// TIA Portal V19 export
FUNCTION_BLOCK "SpeedMachine_FB"   // FB36, LAD
TITLE = OPEN LOOP VELOCITY AXIS WTITH DRIVE S120 DRIVE TEL 1
// stored: Access Published, MemoryReserve 100, SetENOAutomatically false
   VAR_INPUT
      AreaInterface : "AreaInterface";
      ZSI : "udt_ZoneSafetyInterface";
      DSI : "udt_DeviceSafetyInterface";
      Drive : "TAx_DriveInterface";
      DataIn : "SpeedMachine_DataIn";
      CIn : "SpeedMachine_CIn";
      Config : "SpeedMachine_Config";
      HW_ID_TEL1 : HW_SUBMODULE;
   END_VAR
   VAR_OUTPUT
      MachineInterface : "MachineInterface";
      DataOut : "SpeedMachine_DataOut";
      COut : "SpeedMachine_COut";
   END_VAR
   VAR_IN_OUT
      Par : "SpeedMachine_Par";
      Warning : "SpeedMachine_Wng";
      Alarm : "SpeedMachine_Alr";
   END_VAR
   VAR
      Sts : Struct
         Standstill : Bool := TRUE;
         AlarmsPresence : Bool := FALSE;
         WarningsPresence : Bool := FALSE;
         Gen_Cnd : Bool;
         Bwd_Cnd : Bool := FALSE;
         Fwd_Cnd : Bool := FALSE;
         ReductionRatio : LReal := 1.0;   // mm / giro
      END_STRUCT;
      Ctrl : Struct
         StopDueDoorOpeningRequest : Bool;
         StopInPhase : Bool;
         StopProgrammed : Bool;
         StopAborting : Bool;
         Man_HighSpeed : Bool;
         Bwd_Man : Bool;
         Fwd_Man : Bool;
         Bwd_Aut : Bool;
         Fwd_Aut : Bool;
         Fan : Bool;
         Vel : LReal;
         Acc : LReal;
         Dec : LReal;
      END_STRUCT;
      Diag : Struct
         Drive : "TO_Diagnostic";
      END_STRUCT;
      S120 : "SpeedMotor";
      Fan_M : "Motor";
      TON_NoPendingCmd : IEC_TIMER;
      TON_Feed_DelayManChangeSpeed : IEC_TIMER;
      TON_MissingCndBwd { S7_SetPoint := 'True'} : IEC_TIMER;
      TON_MissingCndFwd { S7_SetPoint := 'True'} : IEC_TIMER;
      TON_Fan_DelayOff : IEC_TIMER;
      TON_Brake_TimeOut : IEC_TIMER;
      S120_STW_TEL1 { ExternalAccessible := 'False'; ExternalVisible := 'False'; ExternalWritable := 'False'} : PD_TEL1_IN;
      S120_ZSW_TEL1 { ExternalAccessible := 'False'; ExternalVisible := 'False'; ExternalWritable := 'False'} : PD_TEL1_OUT;
      GETIO_STW_TEL1 { S7_SetPoint := 'True'} : GETIO;
      SETIO_ZSW_TEL1 { S7_SetPoint := 'True'} : SETIO;
      AUX : Struct
         Bwd_Pb : Bool;
         Fwd_Pb : Bool;
      END_STRUCT;
      HMI : Struct
         Sts { S7_SetPoint := 'True'} : "UDT_HMI-Sts_SpeedMachineFB";
      END_STRUCT;
   END_VAR
   VAR_TEMP
      PE : Struct
         Bwd_Pb : Bool;
         Fwd_Pb : Bool;
      END_STRUCT;
      Req : Bool;
      VelMax_EngUnit : LReal;   // mm/min
      AccMax_EngUnit : LReal;   // mm/s²
      DecMax_EngUnit : LReal;   // mm/s²
      StandstillVelocity_RPM : LReal;
   END_VAR
   VAR_TEMP   // added for the SCL form of the ladder/FBD networks
      _w1 : Bool;
      _w2 : Bool;
   END_VAR
BEGIN

REGION Network 1 (SCL): Reset
   IF #AreaInterface.RstAlarms THEN

       #Alarm.BrakeTimeOut :=
       #Alarm.S120_ComErr :=

       #Warning.NotAutReady :=
       #Warning.MissingCnd_Bkw :=
       #Warning.MissingCnd_Fwd := FALSE;
   END_IF;
END_REGION

REGION Network 2: Alarm motor brake timeout
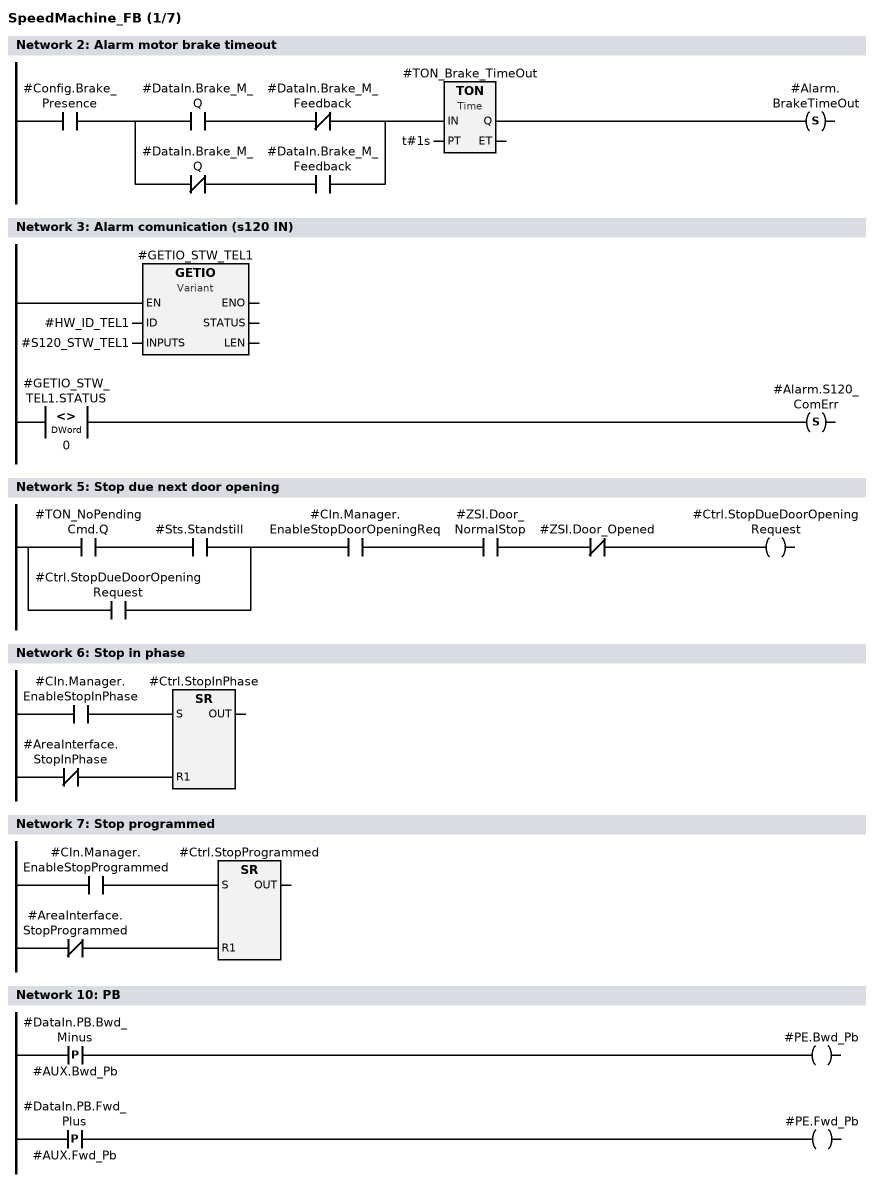
   RUNG wire#powerrail
      Contact( #Config.Brake_Presence )
      wire#w1
      Contact( #DataIn.Brake_M_Q )
      I_Contact( #DataIn.Brake_M_Feedback )
      wire#w2
      { S7_Templates := "time_type := Time" } #TON_Brake_TimeOut.TON(pt := t#1s, et =>)
      S_Coil( #Alarm.BrakeTimeOut )
   END_RUNG
   RUNG wire#w1
      I_Contact( #DataIn.Brake_M_Q )
      Contact( #DataIn.Brake_M_Feedback )
   END_RUNG wire#w2
   // the same network as SCL:
   #TON_Brake_TimeOut.TON(IN := #Config.Brake_Presence AND ((#DataIn.Brake_M_Q AND NOT #DataIn.Brake_M_Feedback) OR (NOT #DataIn.Brake_M_Q AND #DataIn.Brake_M_Feedback)),
                          PT := t#1s);
   IF #TON_Brake_TimeOut.Q THEN #Alarm.BrakeTimeOut := TRUE; END_IF;
END_REGION

REGION Network 3: Alarm comunication (s120 IN)
   RUNG wire#powerrail
      { S7_Templates := "[ptr_type := Variant, id_type := HW_SUBMODULE]" } #GETIO_STW_TEL1.GETIO(ID := #HW_ID_TEL1, INPUTS := #S120_STW_TEL1, STATUS =>, LEN =>)
   END_RUNG
   RUNG wire#powerrail
      { S7_Templates := "SrcType := DWord" } NE_Contact(in1 := #GETIO_STW_TEL1.STATUS, in2 := 0)
      S_Coil( #Alarm.S120_ComErr )
   END_RUNG
   // the same network as SCL:
   #GETIO_STW_TEL1(ID := #HW_ID_TEL1, INPUTS := #S120_STW_TEL1);   // GETIO
   IF #GETIO_STW_TEL1.STATUS <> 0 THEN #Alarm.S120_ComErr := TRUE; END_IF;
END_REGION

REGION Network 4: <<< MACHINE STOP >>>
END_REGION

REGION Network 5: Stop due next door opening
   RUNG wire#powerrail
      Contact( #TON_NoPendingCmd.Q )
      Contact( #Sts.Standstill )
      wire#w1
      Contact( #CIn.Manager.EnableStopDoorOpeningReq )
      Contact( #ZSI.Door_NormalStop )
      I_Contact( #ZSI.Door_Opened )
      Coil( #Ctrl.StopDueDoorOpeningRequest )
   END_RUNG
   RUNG wire#powerrail
      Contact( #Ctrl.StopDueDoorOpeningRequest )
   END_RUNG wire#w1
   // the same network as SCL:
   #Ctrl.StopDueDoorOpeningRequest := ((#TON_NoPendingCmd.Q AND #Sts.Standstill) OR #Ctrl.StopDueDoorOpeningRequest) AND #CIn.Manager.EnableStopDoorOpeningReq AND #ZSI.Door_NormalStop AND NOT #ZSI.Door_Opened;
END_REGION

REGION Network 6: Stop in phase
   RUNG wire#powerrail
      Contact( #CIn.Manager.EnableStopInPhase )
      S_SR(operand := #Ctrl.StopInPhase, r1 := wire#w1)
   END_RUNG
   RUNG wire#powerrail
      I_Contact( #AreaInterface.StopInPhase )
   END_RUNG wire#w1
   // the same network as SCL:
   IF #CIn.Manager.EnableStopInPhase THEN
       #Ctrl.StopInPhase := TRUE;   // SR flip-flop
   END_IF;
   IF NOT #AreaInterface.StopInPhase THEN #Ctrl.StopInPhase := FALSE; END_IF;
END_REGION

REGION Network 7: Stop programmed
   RUNG wire#powerrail
      Contact( #CIn.Manager.EnableStopProgrammed )
      S_SR(operand := #Ctrl.StopProgrammed, r1 := wire#w1)
   END_RUNG
   RUNG wire#powerrail
      I_Contact( #AreaInterface.StopProgrammed )
   END_RUNG wire#w1
   // the same network as SCL:
   IF #CIn.Manager.EnableStopProgrammed THEN
       #Ctrl.StopProgrammed := TRUE;   // SR flip-flop
   END_IF;
   IF NOT #AreaInterface.StopProgrammed THEN #Ctrl.StopProgrammed := FALSE; END_IF;
END_REGION

REGION Network 8: >
END_REGION

REGION Network 9: <<< FEED >>>
END_REGION

REGION Network 10: PB
   RUNG wire#powerrail
      P_Contact(operand := #DataIn.PB.Bwd_Minus, bit := #AUX.Bwd_Pb)
      Coil( #PE.Bwd_Pb )
   END_RUNG
   RUNG wire#powerrail
      P_Contact(operand := #DataIn.PB.Fwd_Plus, bit := #AUX.Fwd_Pb)
      Coil( #PE.Fwd_Pb )
   END_RUNG
   // the same network as SCL:
   #_w1 := #DataIn.PB.Bwd_Minus AND NOT #AUX.Bwd_Pb;   // rising edge of #DataIn.PB.Bwd_Minus
   #AUX.Bwd_Pb := #DataIn.PB.Bwd_Minus;
   #PE.Bwd_Pb := #_w1;
   #_w2 := #DataIn.PB.Fwd_Plus AND NOT #AUX.Fwd_Pb;   // rising edge of #DataIn.PB.Fwd_Plus
   #AUX.Fwd_Pb := #DataIn.PB.Fwd_Plus;
   #PE.Fwd_Pb := #_w2;
END_REGION

REGION Network 11: Man
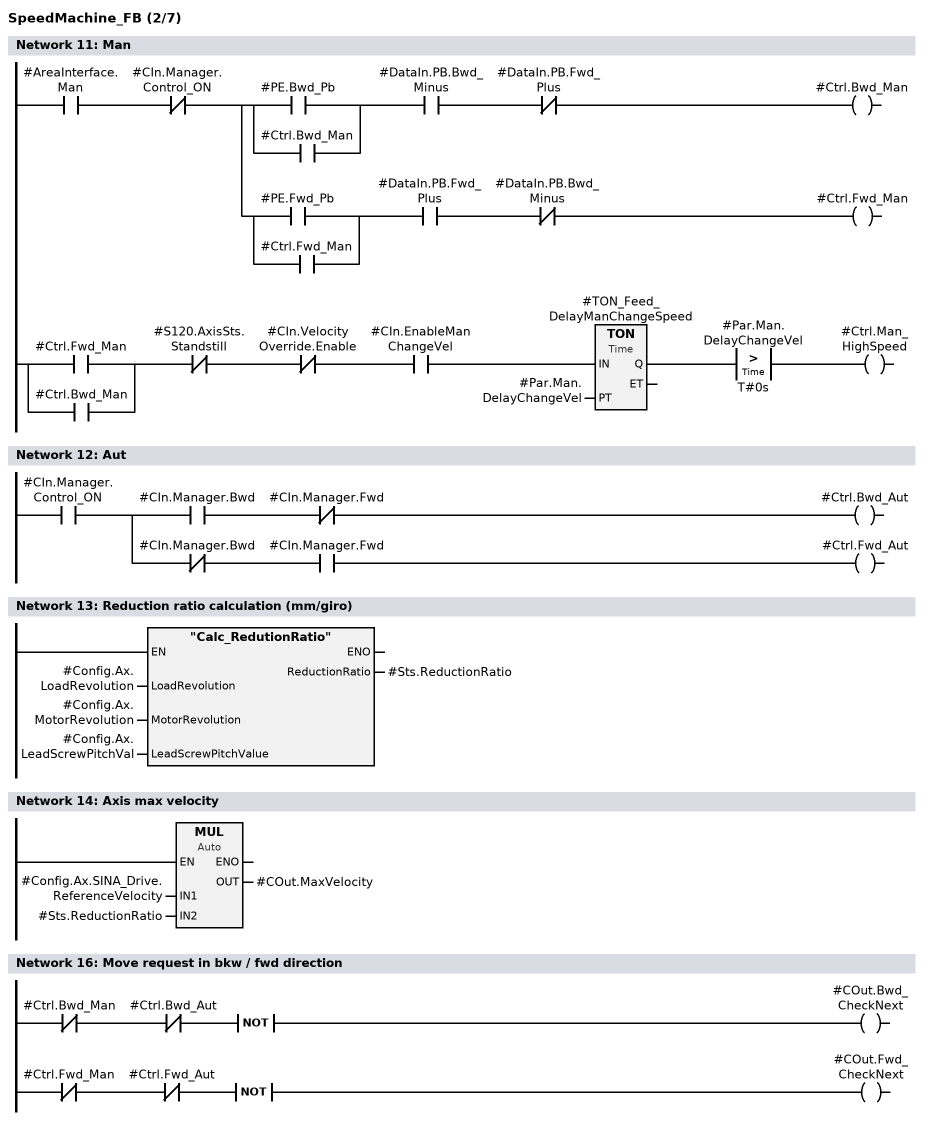
   RUNG wire#powerrail
      Contact( #AreaInterface.Man )
      I_Contact( #CIn.Manager.Control_ON )
      wire#w1
      Contact( #PE.Bwd_Pb )
      wire#w2
      Contact( #DataIn.PB.Bwd_Minus )
      I_Contact( #DataIn.PB.Fwd_Plus )
      Coil( #Ctrl.Bwd_Man )
   END_RUNG
   RUNG wire#w1
      Contact( #Ctrl.Bwd_Man )
   END_RUNG wire#w2
   RUNG wire#w1
      Contact( #PE.Fwd_Pb )
      wire#w3
      Contact( #DataIn.PB.Fwd_Plus )
      I_Contact( #DataIn.PB.Bwd_Minus )
      Coil( #Ctrl.Fwd_Man )
   END_RUNG
   RUNG wire#w1
      Contact( #Ctrl.Fwd_Man )
   END_RUNG wire#w3
   RUNG wire#powerrail
      Contact( #Ctrl.Fwd_Man )
      wire#w4
      I_Contact( #S120.AxisSts.Standstill )
      I_Contact( #CIn.VelocityOverride.Enable )
      Contact( #CIn.EnableManChangeVel )
      { S7_Templates := "time_type := Time" } #TON_Feed_DelayManChangeSpeed.TON(pt := #Par.Man.DelayChangeVel, et =>)
      { S7_Templates := "SrcType := Time" } GT_Contact(in1 := #Par.Man.DelayChangeVel, in2 := T#0s)
      Coil( #Ctrl.Man_HighSpeed )
   END_RUNG
   RUNG wire#powerrail
      Contact( #Ctrl.Bwd_Man )
   END_RUNG wire#w4
   // the same network as SCL:
   #_w1 := #AreaInterface.Man AND NOT #CIn.Manager.Control_ON;
   #Ctrl.Bwd_Man := #_w1 AND (#PE.Bwd_Pb OR #Ctrl.Bwd_Man) AND #DataIn.PB.Bwd_Minus AND NOT #DataIn.PB.Fwd_Plus;
   #Ctrl.Fwd_Man := #_w1 AND (#PE.Fwd_Pb OR #Ctrl.Fwd_Man) AND #DataIn.PB.Fwd_Plus AND NOT #DataIn.PB.Bwd_Minus;
   #TON_Feed_DelayManChangeSpeed.TON(IN := (#Ctrl.Fwd_Man OR #Ctrl.Bwd_Man) AND NOT #S120.AxisSts.Standstill AND NOT #CIn.VelocityOverride.Enable AND #CIn.EnableManChangeVel,
                           PT := #Par.Man.DelayChangeVel);
   #Ctrl.Man_HighSpeed := #TON_Feed_DelayManChangeSpeed.Q AND (#Par.Man.DelayChangeVel > T#0s);
END_REGION

REGION Network 12: Aut
   RUNG wire#powerrail
      Contact( #CIn.Manager.Control_ON )
      wire#w1
      Contact( #CIn.Manager.Bwd )
      I_Contact( #CIn.Manager.Fwd )
      Coil( #Ctrl.Bwd_Aut )
   END_RUNG
   RUNG wire#w1
      I_Contact( #CIn.Manager.Bwd )
      Contact( #CIn.Manager.Fwd )
      Coil( #Ctrl.Fwd_Aut )
   END_RUNG
   // the same network as SCL:
   #Ctrl.Bwd_Aut := #CIn.Manager.Control_ON AND #CIn.Manager.Bwd AND NOT #CIn.Manager.Fwd;
   #Ctrl.Fwd_Aut := #CIn.Manager.Control_ON AND NOT #CIn.Manager.Bwd AND #CIn.Manager.Fwd;
END_REGION

REGION Network 13: Reduction ratio calculation (mm/giro)
   RUNG wire#powerrail
      "Calc_RedutionRatio"(LoadRevolution := #Config.Ax.LoadRevolution, MotorRevolution := #Config.Ax.MotorRevolution, LeadScrewPitchValue := #Config.Ax.LeadScrewPitchVal, ReductionRatio => #Sts.ReductionRatio)
   END_RUNG
   // the same network as SCL:
   "Calc_RedutionRatio"(LoadRevolution := #Config.Ax.LoadRevolution,
                        MotorRevolution := #Config.Ax.MotorRevolution,
                        LeadScrewPitchValue := #Config.Ax.LeadScrewPitchVal,
                        ReductionRatio => #Sts.ReductionRatio);
END_REGION

REGION Network 14: Axis max velocity
   RUNG wire#powerrail
      Mul(in1 := #Config.Ax.SINA_Drive.ReferenceVelocity, in2 := #Sts.ReductionRatio, out => #COut.MaxVelocity)
   END_RUNG
   // the same network as SCL:
   #COut.MaxVelocity := #Config.Ax.SINA_Drive.ReferenceVelocity * #Sts.ReductionRatio;
END_REGION

REGION Network 15 (SCL): Velocity & Dynamics
   #VelMax_EngUnit := #Config.Ax.SINA_Drive.ReferenceVelocity *  #Sts.ReductionRatio;
   #AccMax_EngUnit := (#Config.Ax.SINA_Drive.ReferenceVelocity / 60.0 / #Config.Ax.MinAccTime) * #Sts.ReductionRatio; // Giri/s² * mm/Giro = mm/s²
   #DecMax_EngUnit := (#Config.Ax.SINA_Drive.ReferenceVelocity / 60.0 / #Config.Ax.MinDecTime) * #Sts.ReductionRatio; // Giri/s² * mm/Giro = mm/s²


   #Ctrl.Vel := 0.0;

   IF #Ctrl.Bwd_Man AND #S120.AxisCtrl.MoveMinus THEN


       #Ctrl.Acc := #Par.Man.Acc;
       #Ctrl.Dec := #Par.Man.Dec;

       IF #Ctrl.Man_HighSpeed THEN
           #Ctrl.Vel := #Par.Man.VelBwd;
       ELSE
           #Ctrl.Vel := #Par.Man.VelFwdLow;
       END_IF;

   ELSIF #Ctrl.Fwd_Man AND #S120.AxisCtrl.MovePlus THEN


       #Ctrl.Acc := #Par.Man.Acc;
       #Ctrl.Dec := #Par.Man.Dec;

       IF #Ctrl.Man_HighSpeed THEN
           #Ctrl.Vel := #Par.Man.VelFwdHigh;
       ELSE
           #Ctrl.Vel := #Par.Man.VelFwdLow;
       END_IF;


   ELSIF (#Ctrl.Bwd_Aut AND #S120.AxisCtrl.MoveMinus) OR (#Ctrl.Fwd_Aut AND #S120.AxisCtrl.MovePlus)  THEN

       #Ctrl.Vel := #CIn.Manager.Vel;
       #Ctrl.Acc := #CIn.Manager.Acc;
       #Ctrl.Dec := #CIn.Manager.Dec;

   END_IF;



   // Dynamics limit
   #Ctrl.Vel := MIN(IN1:= #Ctrl.Vel,IN2:= #VelMax_EngUnit);


   #Ctrl.Acc := MIN(IN1:= #Ctrl.Acc,IN2:= #AccMax_EngUnit);

   IF #Ctrl.Acc <= 0.0 THEN
       #Ctrl.Acc := #Par.Man.Acc;
   END_IF;

   #Ctrl.Dec := MIN(IN1:= #Ctrl.Dec,IN2:= #DecMax_EngUnit);
   IF #Ctrl.Dec <= 0.0 THEN
       #Ctrl.Dec := #Par.Man.Dec;
   END_IF;





   // SLS velocity limit
   //
   IF #ZSI.Door_Opened AND #Ctrl.Vel > #Config.SLS_VEL THEN
       #Ctrl.Vel := #Config.SLS_VEL;
   END_IF;


   // Brake not open... Velocity  = 0.0
   // 
   IF #Config.Brake_Presence AND NOT #DataIn.Brake_M_Feedback THEN
       #S120.AxisCtrl.Velocity := 0.0;
   END_IF;



   // Conversion and write dynamics value
   // 
   #S120.AxisCtrl.Velocity := #Ctrl.Vel / #Sts.ReductionRatio; // mm/minuto -> giri/minuto

   // Velocity override
   // 
   IF #CIn.VelocityOverride.Enable THEN

       #S120.AxisCtrl.Velocity := #S120.AxisCtrl.Velocity  * (LIMIT(MN := 1.0, IN := #CIn.VelocityOverride.Value, MX := 200.0)/100);
   END_IF;



   #S120.AxisCtrl.Acceleration := #Ctrl.Acc / #Sts.ReductionRatio; // mm/s2 -> giri/s²
   #S120.AxisCtrl.Deceleration := #Ctrl.Dec / #Sts.ReductionRatio; // mm/s2 -> giri/s²


   //#StandstillVelocity_RPM := #Config.Ax.StandstillVelocity / #Sts.ReductionRatio;
END_REGION

REGION Network 16: Move request in bkw / fwd direction
   RUNG wire#powerrail
      I_Contact( #Ctrl.Bwd_Man )
      I_Contact( #Ctrl.Bwd_Aut )
      Not()
      Coil( #COut.Bwd_CheckNext )
   END_RUNG
   RUNG wire#powerrail
      I_Contact( #Ctrl.Fwd_Man )
      I_Contact( #Ctrl.Fwd_Aut )
      Not()
      Coil( #COut.Fwd_CheckNext )
   END_RUNG
   // the same network as SCL:
   #COut.Bwd_CheckNext := NOT (NOT #Ctrl.Bwd_Man AND NOT #Ctrl.Bwd_Aut);
   #COut.Fwd_CheckNext := NOT (NOT #Ctrl.Fwd_Man AND NOT #Ctrl.Fwd_Aut);
END_REGION

REGION Network 17: Conditions
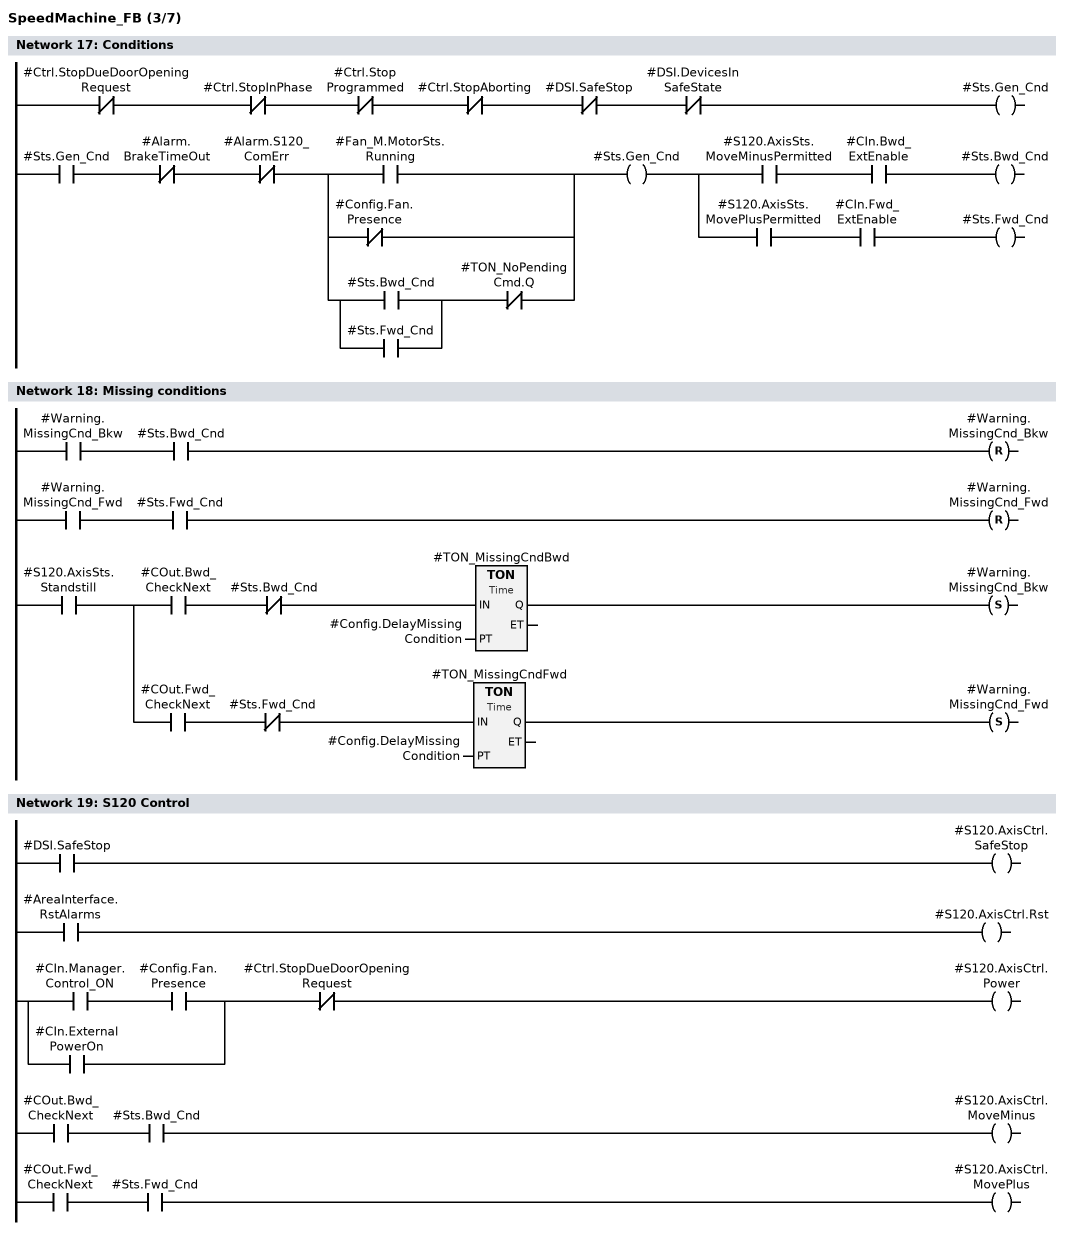
   RUNG wire#powerrail
      I_Contact( #Ctrl.StopDueDoorOpeningRequest )
      I_Contact( #Ctrl.StopInPhase )
      I_Contact( #Ctrl.StopProgrammed )
      I_Contact( #Ctrl.StopAborting )
      I_Contact( #DSI.SafeStop )
      I_Contact( #DSI.DevicesInSafeState )
      Coil( #Sts.Gen_Cnd )
   END_RUNG
   RUNG wire#powerrail
      Contact( #Sts.Gen_Cnd )
      I_Contact( #Alarm.BrakeTimeOut )
      I_Contact( #Alarm.S120_ComErr )
      wire#w1
      Contact( #Fan_M.MotorSts.Running )
      wire#w2
      Coil( #Sts.Gen_Cnd )
      wire#w4
      Contact( #S120.AxisSts.MoveMinusPermitted )
      Contact( #CIn.Bwd_ExtEnable )
      Coil( #Sts.Bwd_Cnd )
   END_RUNG
   RUNG wire#w1
      I_Contact( #Config.Fan.Presence )
   END_RUNG wire#w2
   RUNG wire#w1
      Contact( #Sts.Bwd_Cnd )
      wire#w3
      I_Contact( #TON_NoPendingCmd.Q )
   END_RUNG wire#w2
   RUNG wire#w1
      Contact( #Sts.Fwd_Cnd )
   END_RUNG wire#w3
   RUNG wire#w4
      Contact( #S120.AxisSts.MovePlusPermitted )
      Contact( #CIn.Fwd_ExtEnable )
      Coil( #Sts.Fwd_Cnd )
   END_RUNG
   // the same network as SCL:
   #Sts.Gen_Cnd := NOT #Ctrl.StopDueDoorOpeningRequest AND NOT #Ctrl.StopInPhase AND NOT #Ctrl.StopProgrammed AND NOT #Ctrl.StopAborting AND NOT #DSI.SafeStop AND NOT #DSI.DevicesInSafeState;
   #Sts.Gen_Cnd := #Sts.Gen_Cnd AND NOT #Alarm.BrakeTimeOut AND NOT #Alarm.S120_ComErr AND (#Fan_M.MotorSts.Running OR NOT #Config.Fan.Presence OR ((#Sts.Bwd_Cnd OR #Sts.Fwd_Cnd) AND NOT #TON_NoPendingCmd.Q));
   #Sts.Bwd_Cnd := #Sts.Gen_Cnd AND #S120.AxisSts.MoveMinusPermitted AND #CIn.Bwd_ExtEnable;
   #Sts.Fwd_Cnd := #Sts.Gen_Cnd AND #S120.AxisSts.MovePlusPermitted AND #CIn.Fwd_ExtEnable;
END_REGION

REGION Network 18: Missing conditions
   RUNG wire#powerrail
      Contact( #Warning.MissingCnd_Bkw )
      Contact( #Sts.Bwd_Cnd )
      R_Coil( #Warning.MissingCnd_Bkw )
   END_RUNG
   RUNG wire#powerrail
      Contact( #Warning.MissingCnd_Fwd )
      Contact( #Sts.Fwd_Cnd )
      R_Coil( #Warning.MissingCnd_Fwd )
   END_RUNG
   RUNG wire#powerrail
      Contact( #S120.AxisSts.Standstill )
      wire#w1
      Contact( #COut.Bwd_CheckNext )
      I_Contact( #Sts.Bwd_Cnd )
      { S7_Templates := "time_type := Time" } #TON_MissingCndBwd.TON(pt := #Config.DelayMissingCondition, et =>)
      S_Coil( #Warning.MissingCnd_Bkw )
   END_RUNG
   RUNG wire#w1
      Contact( #COut.Fwd_CheckNext )
      I_Contact( #Sts.Fwd_Cnd )
      { S7_Templates := "time_type := Time" } #TON_MissingCndFwd.TON(pt := #Config.DelayMissingCondition, et =>)
      S_Coil( #Warning.MissingCnd_Fwd )
   END_RUNG
   // the same network as SCL:
   IF #Warning.MissingCnd_Bkw AND #Sts.Bwd_Cnd THEN #Warning.MissingCnd_Bkw := FALSE; END_IF;
   IF #Warning.MissingCnd_Fwd AND #Sts.Fwd_Cnd THEN #Warning.MissingCnd_Fwd := FALSE; END_IF;
   #TON_MissingCndBwd.TON(IN := #S120.AxisSts.Standstill AND #COut.Bwd_CheckNext AND NOT #Sts.Bwd_Cnd,
                          PT := #Config.DelayMissingCondition);
   IF #TON_MissingCndBwd.Q THEN #Warning.MissingCnd_Bkw := TRUE; END_IF;
   #TON_MissingCndFwd.TON(IN := #S120.AxisSts.Standstill AND #COut.Fwd_CheckNext AND NOT #Sts.Fwd_Cnd,
                          PT := #Config.DelayMissingCondition);
   IF #TON_MissingCndFwd.Q THEN #Warning.MissingCnd_Fwd := TRUE; END_IF;
END_REGION

REGION Network 19: S120 Control
   RUNG wire#powerrail
      Contact( #DSI.SafeStop )
      Coil( #S120.AxisCtrl.SafeStop )
   END_RUNG
   RUNG wire#powerrail
      Contact( #AreaInterface.RstAlarms )
      Coil( #S120.AxisCtrl.Rst )
   END_RUNG
   RUNG wire#powerrail
      Contact( #CIn.Manager.Control_ON )
      Contact( #Config.Fan.Presence )
      wire#w1
      I_Contact( #Ctrl.StopDueDoorOpeningRequest )
      Coil( #S120.AxisCtrl.Power )
   END_RUNG
   RUNG wire#powerrail
      Contact( #CIn.ExternalPowerOn )
   END_RUNG wire#w1
   RUNG wire#powerrail
      Contact( #COut.Bwd_CheckNext )
      Contact( #Sts.Bwd_Cnd )
      Coil( #S120.AxisCtrl.MoveMinus )
   END_RUNG
   RUNG wire#powerrail
      Contact( #COut.Fwd_CheckNext )
      Contact( #Sts.Fwd_Cnd )
      Coil( #S120.AxisCtrl.MovePlus )
   END_RUNG
   // the same network as SCL:
   #S120.AxisCtrl.SafeStop := #DSI.SafeStop;
   #S120.AxisCtrl.Rst := #AreaInterface.RstAlarms;
   #S120.AxisCtrl.Power := ((#CIn.Manager.Control_ON AND #Config.Fan.Presence) OR #CIn.ExternalPowerOn) AND NOT #Ctrl.StopDueDoorOpeningRequest;
   #S120.AxisCtrl.MoveMinus := #COut.Bwd_CheckNext AND #Sts.Bwd_Cnd;
   #S120.AxisCtrl.MovePlus := #COut.Fwd_CheckNext AND #Sts.Fwd_Cnd;
END_REGION

REGION Network 20: S120 manager
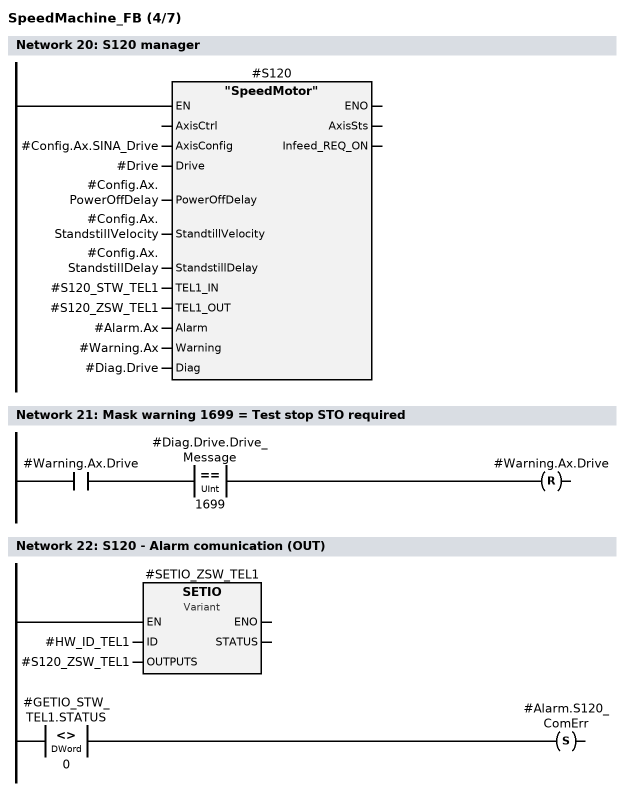
   RUNG wire#powerrail
      #S120(AxisCtrl :=, AxisConfig := #Config.Ax.SINA_Drive, Drive := #Drive, PowerOffDelay := #Config.Ax.PowerOffDelay, StandtillVelocity := #Config.Ax.StandstillVelocity, StandstillDelay := #Config.Ax.StandstillDelay, TEL1_IN := #S120_STW_TEL1, TEL1_OUT := #S120_ZSW_TEL1, Alarm := #Alarm.Ax, Warning := #Warning.Ax, Diag := #Diag.Drive, AxisSts =>, Infeed_REQ_ON =>)
   END_RUNG
   // the same network as SCL:
   #S120(AxisConfig := #Config.Ax.SINA_Drive,   // "SpeedMotor"
         Drive := #Drive,
         PowerOffDelay := #Config.Ax.PowerOffDelay,
         StandtillVelocity := #Config.Ax.StandstillVelocity,
         StandstillDelay := #Config.Ax.StandstillDelay,
         TEL1_IN := #S120_STW_TEL1,
         TEL1_OUT := #S120_ZSW_TEL1,
         Alarm := #Alarm.Ax,
         Warning := #Warning.Ax,
         Diag := #Diag.Drive);
END_REGION

REGION Network 21: Mask warning 1699 = Test stop STO required
   RUNG wire#powerrail
      Contact( #Warning.Ax.Drive )
      { S7_Templates := "SrcType := UInt" } EQ_Contact(in1 := #Diag.Drive.Drive_Message, in2 := 1699)
      R_Coil( #Warning.Ax.Drive )
   END_RUNG
   // the same network as SCL:
   IF #Warning.Ax.Drive AND (#Diag.Drive.Drive_Message = 1699) THEN #Warning.Ax.Drive := FALSE; END_IF;
END_REGION

REGION Network 22: S120 - Alarm comunication (OUT)
   RUNG wire#powerrail
      { S7_Templates := "[card := 0, ptr_type := Variant, id_type := HW_SUBMODULE]" } #SETIO_ZSW_TEL1.SETIO(ID := #HW_ID_TEL1, OUTPUTS := #S120_ZSW_TEL1, STATUS =>)
   END_RUNG
   RUNG wire#powerrail
      { S7_Templates := "SrcType := DWord" } NE_Contact(in1 := #GETIO_STW_TEL1.STATUS, in2 := 0)
      S_Coil( #Alarm.S120_ComErr )
   END_RUNG
   // the same network as SCL:
   #SETIO_ZSW_TEL1(ID := #HW_ID_TEL1, OUTPUTS := #S120_ZSW_TEL1);   // SETIO
   IF #GETIO_STW_TEL1.STATUS <> 0 THEN #Alarm.S120_ComErr := TRUE; END_IF;
END_REGION

REGION Network 23: Coordination Out
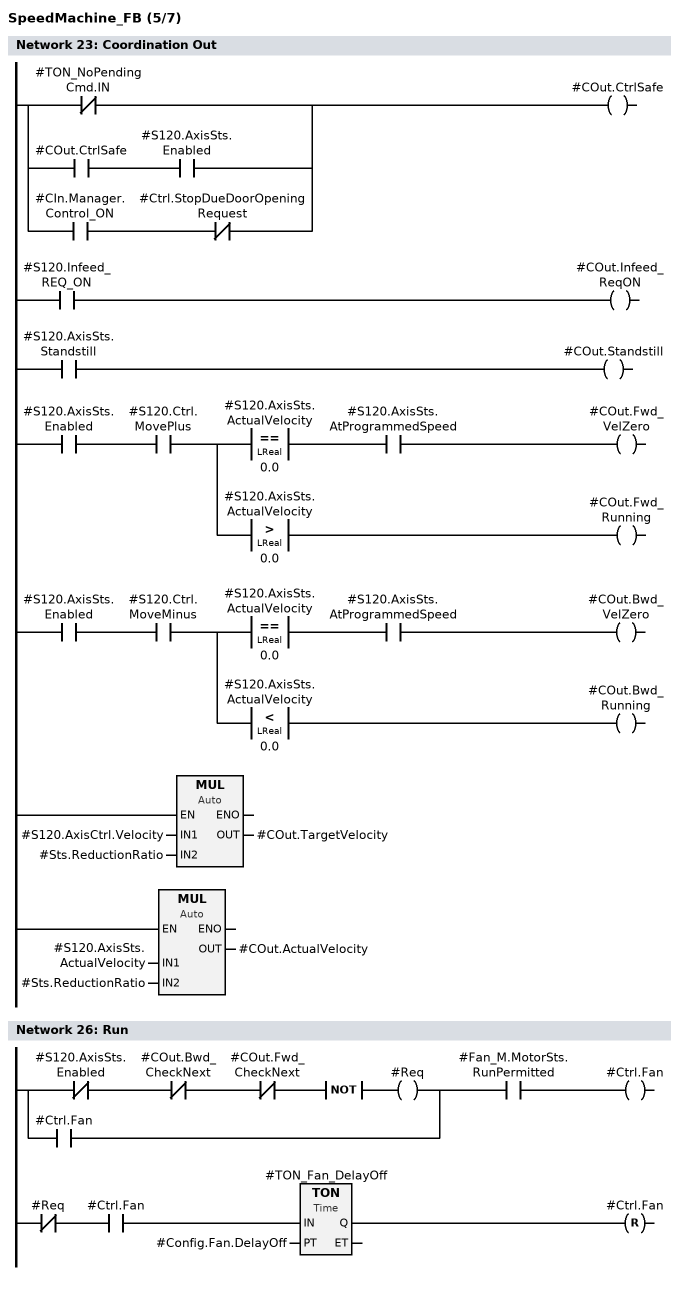
   RUNG wire#powerrail
      I_Contact( #TON_NoPendingCmd.IN )
      wire#w1
      Coil( #COut.CtrlSafe )
   END_RUNG
   RUNG wire#powerrail
      Contact( #COut.CtrlSafe )
      Contact( #S120.AxisSts.Enabled )
   END_RUNG wire#w1
   RUNG wire#powerrail
      Contact( #CIn.Manager.Control_ON )
      I_Contact( #Ctrl.StopDueDoorOpeningRequest )
   END_RUNG wire#w1
   RUNG wire#powerrail
      Contact( #S120.Infeed_REQ_ON )
      Coil( #COut.Infeed_ReqON )
   END_RUNG
   RUNG wire#powerrail
      Contact( #S120.AxisSts.Standstill )
      Coil( #COut.Standstill )
   END_RUNG
   RUNG wire#powerrail
      Contact( #S120.AxisSts.Enabled )
      Contact( #S120.Ctrl.MovePlus )
      wire#w2
      { S7_Templates := "SrcType := LReal" } EQ_Contact(in1 := #S120.AxisSts.ActualVelocity, in2 := 0.0)
      Contact( #S120.AxisSts.AtProgrammedSpeed )
      Coil( #COut.Fwd_VelZero )
   END_RUNG
   RUNG wire#w2
      { S7_Templates := "SrcType := LReal" } GT_Contact(in1 := #S120.AxisSts.ActualVelocity, in2 := 0.0)
      Coil( #COut.Fwd_Running )
   END_RUNG
   RUNG wire#powerrail
      Contact( #S120.AxisSts.Enabled )
      Contact( #S120.Ctrl.MoveMinus )
      wire#w3
      { S7_Templates := "SrcType := LReal" } EQ_Contact(in1 := #S120.AxisSts.ActualVelocity, in2 := 0.0)
      Contact( #S120.AxisSts.AtProgrammedSpeed )
      Coil( #COut.Bwd_VelZero )
   END_RUNG
   RUNG wire#w3
      { S7_Templates := "SrcType := LReal" } LT_Contact(in1 := #S120.AxisSts.ActualVelocity, in2 := 0.0)
      Coil( #COut.Bwd_Running )
   END_RUNG
   RUNG wire#powerrail
      { S7_GenerateENO := "TRUE" } Mul(in1 := #S120.AxisCtrl.Velocity, in2 := #Sts.ReductionRatio, out => #COut.TargetVelocity)
   END_RUNG
   RUNG wire#powerrail
      { S7_GenerateENO := "TRUE" } Mul(in1 := #S120.AxisSts.ActualVelocity, in2 := #Sts.ReductionRatio, out => #COut.ActualVelocity)
   END_RUNG
   // the same network as SCL:
   #COut.CtrlSafe := NOT #TON_NoPendingCmd.IN OR (#COut.CtrlSafe AND #S120.AxisSts.Enabled) OR (#CIn.Manager.Control_ON AND NOT #Ctrl.StopDueDoorOpeningRequest);
   #COut.Infeed_ReqON := #S120.Infeed_REQ_ON;
   #COut.Standstill := #S120.AxisSts.Standstill;
   #_w1 := #S120.AxisSts.Enabled AND #S120.Ctrl.MovePlus;
   #COut.Fwd_VelZero := #_w1 AND (#S120.AxisSts.ActualVelocity = 0.0) AND #S120.AxisSts.AtProgrammedSpeed;
   #COut.Fwd_Running := #_w1 AND (#S120.AxisSts.ActualVelocity > 0.0);
   #_w2 := #S120.AxisSts.Enabled AND #S120.Ctrl.MoveMinus;
   #COut.Bwd_VelZero := #_w2 AND (#S120.AxisSts.ActualVelocity = 0.0) AND #S120.AxisSts.AtProgrammedSpeed;
   #COut.Bwd_Running := #_w2 AND (#S120.AxisSts.ActualVelocity < 0.0);
   #COut.TargetVelocity := #S120.AxisCtrl.Velocity * #Sts.ReductionRatio;
   #COut.ActualVelocity := #S120.AxisSts.ActualVelocity * #Sts.ReductionRatio;
END_REGION

REGION Network 24: >
END_REGION

REGION Network 25: <<< MOTOR FAN >>>
END_REGION

REGION Network 26: Run
   RUNG wire#powerrail
      I_Contact( #S120.AxisSts.Enabled )
      I_Contact( #COut.Bwd_CheckNext )
      I_Contact( #COut.Fwd_CheckNext )
      Not()
      Coil( #Req )
      wire#w1
      Contact( #Fan_M.MotorSts.RunPermitted )
      Coil( #Ctrl.Fan )
   END_RUNG
   RUNG wire#powerrail
      Contact( #Ctrl.Fan )
   END_RUNG wire#w1
   RUNG wire#powerrail
      I_Contact( #Req )
      Contact( #Ctrl.Fan )
      { S7_Templates := "time_type := Time" } #TON_Fan_DelayOff.TON(pt := #Config.Fan.DelayOff, et =>)
      R_Coil( #Ctrl.Fan )
   END_RUNG
   // the same network as SCL:
   #Req := NOT (NOT #S120.AxisSts.Enabled AND NOT #COut.Bwd_CheckNext AND NOT #COut.Fwd_CheckNext);
   #Ctrl.Fan := (#Req OR #Ctrl.Fan) AND #Fan_M.MotorSts.RunPermitted;
   #TON_Fan_DelayOff.TON(IN := NOT #Req AND #Ctrl.Fan, PT := #Config.Fan.DelayOff);
   IF #TON_Fan_DelayOff.Q THEN #Ctrl.Fan := FALSE; END_IF;
END_REGION

REGION Network 27: Device
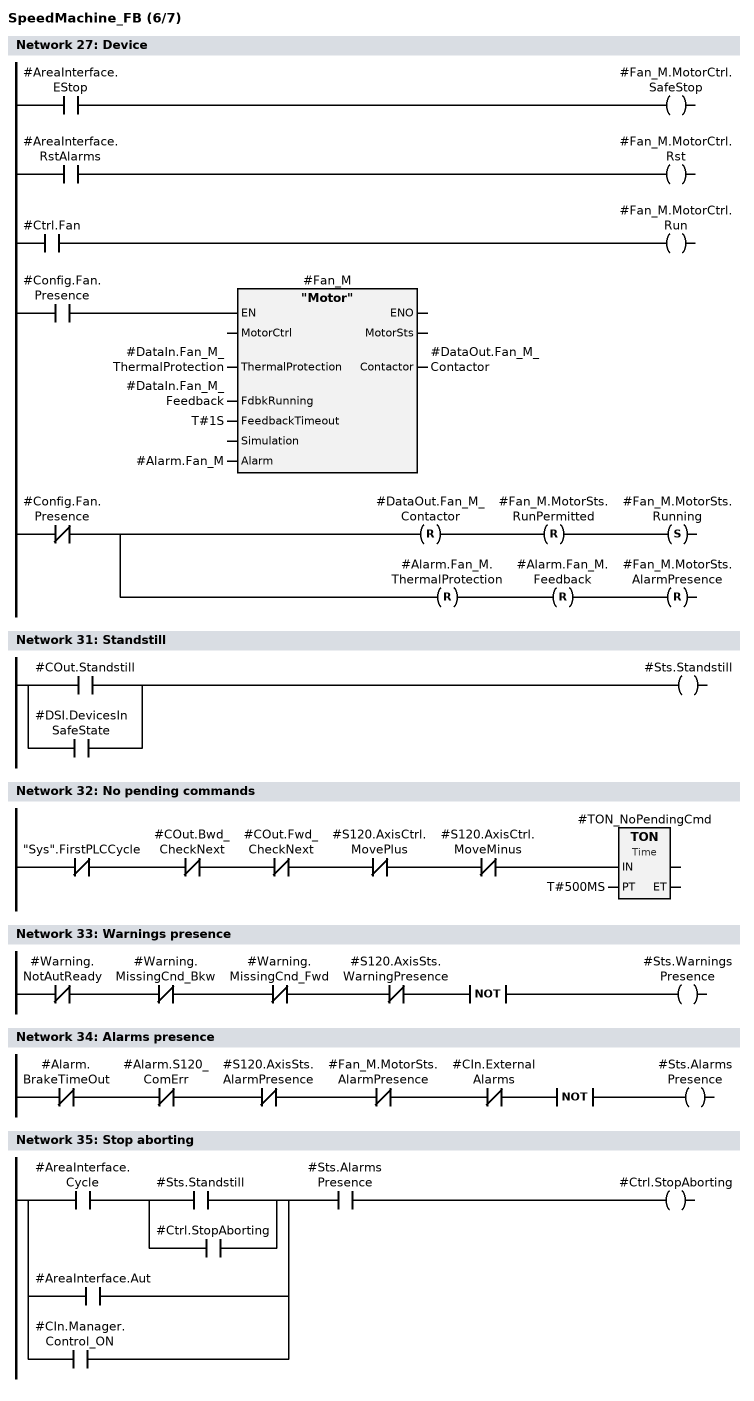
   RUNG wire#powerrail
      Contact( #AreaInterface.EStop )
      Coil( #Fan_M.MotorCtrl.SafeStop )
   END_RUNG
   RUNG wire#powerrail
      Contact( #AreaInterface.RstAlarms )
      Coil( #Fan_M.MotorCtrl.Rst )
   END_RUNG
   RUNG wire#powerrail
      Contact( #Ctrl.Fan )
      Coil( #Fan_M.MotorCtrl.Run )
   END_RUNG
   RUNG wire#powerrail
      Contact( #Config.Fan.Presence )
      #Fan_M(MotorCtrl :=, ThermalProtection := #DataIn.Fan_M_ThermalProtection, FdbkRunning := #DataIn.Fan_M_Feedback, FeedbackTimeout := T#1S, Simulation :=, Alarm := #Alarm.Fan_M, MotorSts =>, Contactor => #DataOut.Fan_M_Contactor)
   END_RUNG
   RUNG wire#powerrail
      I_Contact( #Config.Fan.Presence )
      wire#w1
      R_Coil( #DataOut.Fan_M_Contactor )
      R_Coil( #Fan_M.MotorSts.RunPermitted )
      S_Coil( #Fan_M.MotorSts.Running )
   END_RUNG
   RUNG wire#w1
      R_Coil( #Alarm.Fan_M.ThermalProtection )
      R_Coil( #Alarm.Fan_M.Feedback )
      R_Coil( #Fan_M.MotorSts.AlarmPresence )
   END_RUNG
   // the same network as SCL:
   #Fan_M.MotorCtrl.SafeStop := #AreaInterface.EStop;
   #Fan_M.MotorCtrl.Rst := #AreaInterface.RstAlarms;
   #Fan_M.MotorCtrl.Run := #Ctrl.Fan;
   IF #Config.Fan.Presence THEN
       #Fan_M(ThermalProtection := #DataIn.Fan_M_ThermalProtection,   // "Motor"
              FdbkRunning := #DataIn.Fan_M_Feedback,
              FeedbackTimeout := T#1S,
              Alarm := #Alarm.Fan_M,
              Contactor => #DataOut.Fan_M_Contactor);
   END_IF;
   IF NOT #Config.Fan.Presence THEN
       #DataOut.Fan_M_Contactor := FALSE;
       #Fan_M.MotorSts.RunPermitted := FALSE;
       #Fan_M.MotorSts.Running := TRUE;
       #Alarm.Fan_M.ThermalProtection := FALSE;
       #Alarm.Fan_M.Feedback := FALSE;
       #Fan_M.MotorSts.AlarmPresence := FALSE;
   END_IF;
END_REGION

REGION Network 28: >
END_REGION

REGION Network 29: >
END_REGION

REGION Network 30: <<< MACHINE STATUS >>>
END_REGION

REGION Network 31: Standstill
   RUNG wire#powerrail
      Contact( #COut.Standstill )
      wire#w1
      Coil( #Sts.Standstill )
   END_RUNG
   RUNG wire#powerrail
      Contact( #DSI.DevicesInSafeState )
   END_RUNG wire#w1
   // the same network as SCL:
   #Sts.Standstill := #COut.Standstill OR #DSI.DevicesInSafeState;
END_REGION

REGION Network 32: No pending commands
   RUNG wire#powerrail
      I_Contact( "Sys".FirstPLCCycle )
      I_Contact( #COut.Bwd_CheckNext )
      I_Contact( #COut.Fwd_CheckNext )
      I_Contact( #S120.AxisCtrl.MovePlus )
      I_Contact( #S120.AxisCtrl.MoveMinus )
      { S7_Templates := "time_type := Time" } #TON_NoPendingCmd.TON(pt := T#500MS, et =>)
   END_RUNG
   // the same network as SCL:
   #TON_NoPendingCmd.TON(IN := NOT "Sys".FirstPLCCycle AND NOT #COut.Bwd_CheckNext AND NOT #COut.Fwd_CheckNext AND NOT #S120.AxisCtrl.MovePlus AND NOT #S120.AxisCtrl.MoveMinus,
                         PT := T#500MS);
END_REGION

REGION Network 33: Warnings presence
   RUNG wire#powerrail
      I_Contact( #Warning.NotAutReady )
      I_Contact( #Warning.MissingCnd_Bkw )
      I_Contact( #Warning.MissingCnd_Fwd )
      I_Contact( #S120.AxisSts.WarningPresence )
      Not()
      Coil( #Sts.WarningsPresence )
   END_RUNG
   // the same network as SCL:
   #Sts.WarningsPresence := NOT (NOT #Warning.NotAutReady AND NOT #Warning.MissingCnd_Bkw AND NOT #Warning.MissingCnd_Fwd AND NOT #S120.AxisSts.WarningPresence);
END_REGION

REGION Network 34: Alarms presence
   RUNG wire#powerrail
      I_Contact( #Alarm.BrakeTimeOut )
      I_Contact( #Alarm.S120_ComErr )
      I_Contact( #S120.AxisSts.AlarmPresence )
      I_Contact( #Fan_M.MotorSts.AlarmPresence )
      I_Contact( #CIn.ExternalAlarms )
      Not()
      Coil( #Sts.AlarmsPresence )
   END_RUNG
   // the same network as SCL:
   #Sts.AlarmsPresence := NOT (NOT #Alarm.BrakeTimeOut AND NOT #Alarm.S120_ComErr AND NOT #S120.AxisSts.AlarmPresence AND NOT #Fan_M.MotorSts.AlarmPresence AND NOT #CIn.ExternalAlarms);
END_REGION

REGION Network 35: Stop aborting
   RUNG wire#powerrail
      Contact( #AreaInterface.Cycle )
      wire#w1
      Contact( #Sts.Standstill )
      wire#w2
      Contact( #Sts.AlarmsPresence )
      Coil( #Ctrl.StopAborting )
   END_RUNG
   RUNG wire#w1
      Contact( #Ctrl.StopAborting )
   END_RUNG wire#w2
   RUNG wire#powerrail
      Contact( #AreaInterface.Aut )
   END_RUNG wire#w2
   RUNG wire#powerrail
      Contact( #CIn.Manager.Control_ON )
   END_RUNG wire#w2
   // the same network as SCL:
   #Ctrl.StopAborting := ((#AreaInterface.Cycle AND (#Sts.Standstill OR #Ctrl.StopAborting)) OR #AreaInterface.Aut OR #CIn.Manager.Control_ON) AND #Sts.AlarmsPresence;
END_REGION

REGION Network 36 (SCL): Collect machine to zone interface
   #MachineInterface.AutReady := #AreaInterface.Aut AND NOT #Sts.AlarmsPresence;
   #MachineInterface.Aborting := #Ctrl.StopAborting;
   #MachineInterface.MotionsStandStill := #TON_NoPendingCmd.Q AND #Sts.Standstill;
   #MachineInterface.AckStopInPhase := #Ctrl.StopInPhase AND #MachineInterface.MotionsStandStill;
   #MachineInterface.AckStopProgrammed := #Ctrl.StopProgrammed AND #MachineInterface.MotionsStandStill;
   #MachineInterface.AlarmsPresence := #Sts.AlarmsPresence;
   #MachineInterface.WarningPresence := #Sts.WarningsPresence;
END_REGION

REGION Network 37: Warning Machine not ready for automatic
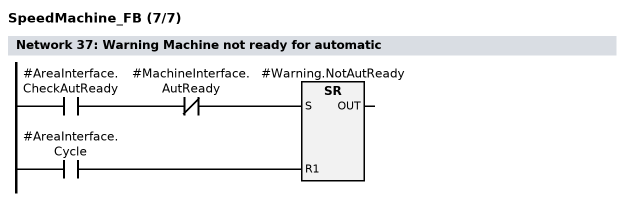
   RUNG wire#powerrail
      Contact( #AreaInterface.CheckAutReady )
      I_Contact( #MachineInterface.AutReady )
      S_SR(operand := #Warning.NotAutReady, r1 := wire#w1)
   END_RUNG
   RUNG wire#powerrail
      Contact( #AreaInterface.Cycle )
   END_RUNG wire#w1
   // the same network as SCL:
   IF #AreaInterface.CheckAutReady AND NOT #MachineInterface.AutReady THEN
       #Warning.NotAutReady := TRUE;   // SR flip-flop
   END_IF;
   IF #AreaInterface.Cycle THEN #Warning.NotAutReady := FALSE; END_IF;
END_REGION

REGION Network 38: >
END_REGION

REGION Network 39 (SCL): HMI Status SpeedMachine
   // Area dati Status per HMI sull'azionamento

   #HMI.Sts.Enabled := #S120.AxisSts.Enabled;
   #HMI.Sts.Standstill := #Sts.Standstill;
   #HMI.Sts.Frw_Run := #COut.Fwd_Running;
   #HMI.Sts.Bwd_Run := #COut.Bwd_Running;
   #HMI.Sts.Alarm := #Sts.AlarmsPresence;
   #HMI.Sts.Warning := #Sts.WarningsPresence;
   #HMI.Sts.Target_Vel := #Ctrl.Vel;
   #HMI.Sts.Actual_Vel := #COut.ActualVelocity;
END_REGION

REGION Network 40: >
END_REGION
END_FUNCTION_BLOCK
